INTERFACE I_Module EXTENDS I_ContainComponents, I_ContainModules, I_Base

METHOD Accept
VAR_INPUT
	Visitor : I_ModuleVisitor;
END_VAR
END_METHOD

METHOD DeregisterWithParent
VAR_INPUT
	Parent : I_ContainModules;
END_VAR
END_METHOD

{attribute 'monitoring' := 'call'}
PROPERTY Name : T_MaxString
GET
END_GET
END_PROPERTY

METHOD RegisterWithParent
VAR_INPUT
	Parent : I_ContainModules;
END_VAR
END_METHOD

METHOD ResetComponents : BOOL
END_METHOD

METHOD ResetModules : BOOL
END_METHOD

END_INTERFACE

(* stored: Version 1.1.0.1, ProductVersion 3.1.4026.18
   Itf I_Module: Id {abdc2707-eea5-4b43-9b07-7c9c593bb60d}
   Method Accept: Id {ed2f01ce-0901-480b-b14f-5f4ea8dd406d}
   Method DeregisterWithParent: Id {85e7f18d-e30e-436d-88cc-cfcd0938a84b}
   Property Name: Id {645dead5-ca4e-489b-a742-ccdef1b7fc18}
   Get Get: Id {54e077c2-cb3e-43c2-b722-968bb81d61c6}
   Method RegisterWithParent: Id {9377ff83-3c4e-440d-9f12-20e3c4e37115}
   Method ResetComponents: Id {b058bb8f-c663-4af3-a6e2-40a7aeaa18db}
   Method ResetModules: Id {ab9c2664-14e8-4ad8-af34-4e0b3e2ab838} *)
